// TIA Portal project "Tanque_PID" (V16)

(* hardware
DEVICE "S71500/ET200MP station_1"  S7-1500 station
   slot 0: "Perfil soporte_0"  Rack  6ES7 590-1***0-0AA0
   slot 1: "PLC_1"  CPU 1511-1 PN  6ES7 511-1AK02-0AB0  V2.5
      slot 3: "Display de la CPU_1"  6ES7591-1AA00-0AA0
      slot 32768: "Interfaz PROFINET_1"  X1
         slot 32769: "Puerto_1"  X1 P1
         slot 32770: "Puerto_2"  X1 P2
DEVICE "PC-System_1"  SIMATIC PC station
   slot 0: "Estación PC SIMATIC"  Rail  SIMATIC PC-Station  V1.0
      slot 125: "Stationmanager"  Station_Manager  V6.0.4
   slot 1: "HMI_RT_1"  WinCC RT Advanced  6AV2 104-0xxxx-xxxx  16.0.0.0
      slot 33792: "Interfaz del equipo"  Host interface
   slot 2: "IE general_1"  IE General  IE_CP  V8.2.0
*)

// ===== PLC "PLC_1"  CPU 1511-1 PN =====

VAR_GLOBAL   // PLC tag table "Tabla de variables estándar"
   "START_SISTEMA" AT %I0.0 : Bool;
   "STOP_SISTEMA" AT %I0.1 : Bool;
   "ENCENDIDO_SISTEMA" AT %M1.0 : Bool;
   "START_LIGHT" AT %Q0.0 : Bool;
   "STOP_LIGTH" AT %Q0.1 : Bool;
   "FILL_VALVE" AT %QW100 : Word;
   "DISCHARGE_VALVE" AT %QW102 : Word;
   "INPUT_FILL_VALVE" AT %MW10 : Word;
   "INPUT_DISCHARGE_VALVE" AT %MW12 : Word;
   "INPUT_FILL_VALVE_NORMAL" AT %MD14 : Real;
   "INPUT_DICHARGE_VALVE_NORMAL" AT %MD18 : Real;
   "DATA_INPUT_FILL_VALVE" AT %MW22 : Word;
   "DATA_INPUT_DISCHARGE_VALVE" AT %MW24 : Word;
   "CONTROL_MANUAL" AT %M1.1 : Bool;
   "CONTROL_AUTOMATICO_PID" AT %M1.2 : Bool;
   "LEVEL_METER" AT %IW100 : Word;
   "LEVEL_METER_NORMAL" AT %MD28 : Real;
   "LEVEL_METER_PANTALLA" AT %QW106 : Word;
   "INPUT_SP" AT %MW32 : Word;
   "SP_PANTALLA" AT %QW104 : Word;
   "SENSOR_NIVEL_INFERIOR" AT %I0.2 : Bool;
   "SENSOR_NIVEL_SUPERIOR" AT %I0.3 : Bool;
   "TANQUE_VACIO" AT %Q0.2 : Bool;
   "TANQUE_LLENO" AT %Q0.3 : Bool;
   "ON_PID_NIVEL" AT %M1.3 : Bool;
   "OFF_PID_NIVEL" AT %M1.4 : Bool;
   "PID_NIVEL" AT %M1.5 : Bool;
   "ON_PID_MANUAL" AT %M1.6 : Bool;
   "OFF_PID_MANUAL" AT %M1.7 : Bool;
   "PID_SET_MANUAL" AT %M2.0 : Bool;
   "DATA_PID_GAIN" AT %MD34 : Real;
   "DATA_PID_TI" AT %MD38 : Real;
   "DATA_PID_TD" AT %MD42 : Real;
   "OUT_PID_FILL_VALVE" AT %MW46 : Word;
   "INPUT_SP_PID" AT %MD48 : Real;
   "LEVEL_METER_PID" AT %MD54 : Real;
   "OUT_PID_FILL_VALVE_PID" AT %MD60 : Real;
   "START_SISTEMA_HMI" AT %M2.2 : Bool;
   "STOP_SISTEMA_HMI" AT %M2.3 : Bool;
   "CONTROL_MANUAL_CAUDAL" AT %M2.4 : Bool;
   "CONTROL_AUTOMATICO_PID_CAUDAL" AT %M2.5 : Bool;
   "CAUDAL_METER" AT %IW104 : Word;
   "CAUDAL_METER_NORMAL" AT %MD64 : Real;
   "CAUDAL_METER_PANTALLA" AT %QW110 : Word;
   "INPUT_SP_CAUDAL" AT %MW68 : Word;
   "SP_PANTALLA_CAUDAL" AT %QW112 : Word;
   "ON_PID_CAUDAL" AT %M2.6 : Bool;
   "OFF_PID_CAUDAL" AT %M2.7 : Bool;
   "PID_SET_MANUAL_CAUDAL" AT %M3.0 : Bool;
   "DATA_PID_GAIN_CAUDAL" AT %MD70 : Real;
   "DATA_PID_TI_CAUDAL" AT %MD74 : Real;
   "DATA_PID_TD_CAUDAL" AT %MD76 : Real;
   "INPUT_SP_PID_CAUDAL" AT %MD80 : Real;
   "CAUDAL_METER_PID" AT %MD84 : Real;
   "SENSOR_CAUDAL" AT %ID88 : Real;
   "OUT_PID_DISCHARGE_VALVE" AT %MW114 : Word;
   "OUT_PID_DISCHARGE_VALVE_PID" AT %MD92 : Real;
   "PID_CAUDAL" AT %M3.1 : Bool;
   "ON_PID_MANUAL_CAUDAL" AT %M3.2 : Bool;
   "OFF_PID_MANUAL_CAUDAL" AT %M3.3 : Bool;
   "PID_OUTPUT" AT %MD96 : Real;
   "ABS_PID_OUTPUT" AT %MD100 : Real;
   "SP_PANTALLA_MAS" AT %QW116 : Word;
   "SP_PANTALLA_MENOs" AT %QW118 : Word;
   "MITAD_VALVULA" AT %MD104 : Real;
   "50_VALVULA" AT %MW118 : Word;
   "PORCENT_CONEXION" AT %MD108 : Real;
   "PORCENT_NIVEL" AT %MD120 : Real;
   "PORCENT_NIVEL_INT" AT %MW122 : Word;
END_VAR

ORGANIZATION_BLOCK "1_Main"   // OB1, LAD, ProgramCycle
TITLE = "Main Program Sweep (Cycle)"
{ S7_Optimized_Access := 'TRUE' }
VERSION : 0.1
   VAR_INPUT
      Initial_Call : Bool;   // Initial call of this OB
      Remanence : Bool;   // =True, if remanent data are available
   END_VAR
   VAR_TEMP   // added for the SCL form of the ladder/FBD networks
      _w1 : Bool;
      _w2 : Bool;
      _w3 : Bool;
   END_VAR
BEGIN

REGION Network 1: ENCENDIDO Y APAGADO DEL SISTEMA
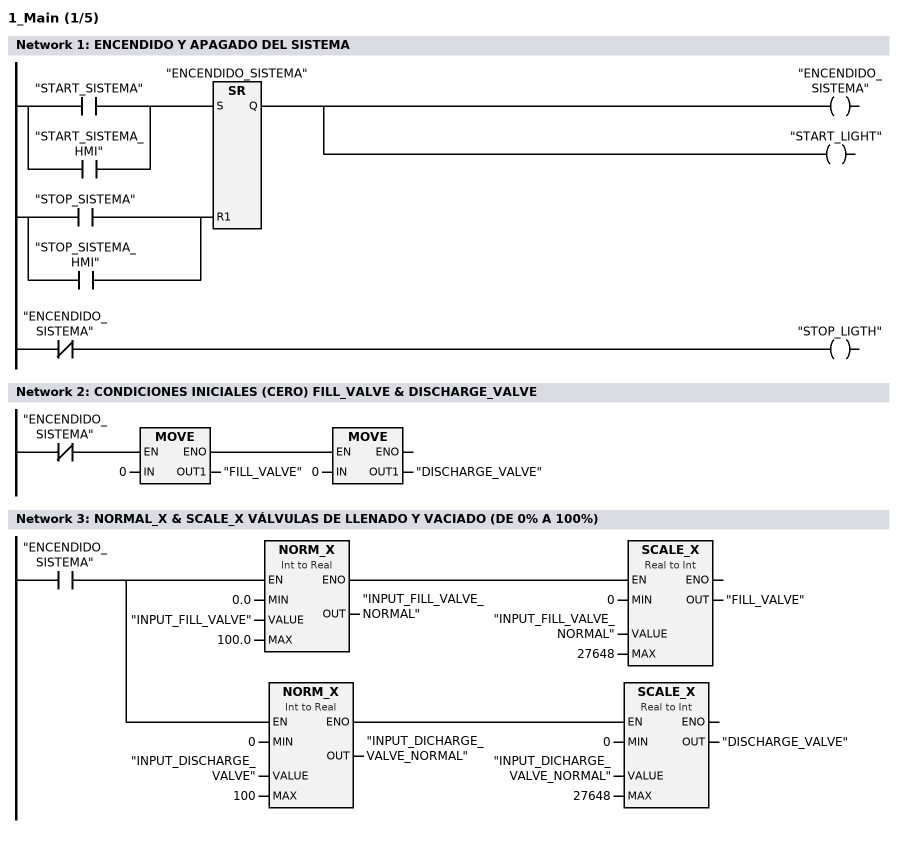
   RUNG wire#powerrail
      Contact( "START_SISTEMA" )
      wire#w1
      S_SR(operand := "ENCENDIDO_SISTEMA", r1 := wire#w2)
      wire#w3
      Coil( "ENCENDIDO_SISTEMA" )
   END_RUNG
   RUNG wire#powerrail
      Contact( "START_SISTEMA_HMI" )
   END_RUNG wire#w1
   RUNG wire#powerrail
      Contact( "STOP_SISTEMA" )
   END_RUNG wire#w2
   RUNG wire#powerrail
      Contact( "STOP_SISTEMA_HMI" )
   END_RUNG wire#w2
   RUNG wire#w3
      Coil( "START_LIGHT" )
   END_RUNG
   RUNG wire#powerrail
      I_Contact( "ENCENDIDO_SISTEMA" )
      Coil( "STOP_LIGTH" )
   END_RUNG
   // the same network as SCL:
   IF "START_SISTEMA" OR "START_SISTEMA_HMI" THEN
       "ENCENDIDO_SISTEMA" := TRUE;   // SR flip-flop
   END_IF;
   IF "STOP_SISTEMA" OR "STOP_SISTEMA_HMI" THEN "ENCENDIDO_SISTEMA" := FALSE; END_IF;
   #_w1 := "ENCENDIDO_SISTEMA";
   "ENCENDIDO_SISTEMA" := "ENCENDIDO_SISTEMA";
   "START_LIGHT" := #_w1;
   "STOP_LIGTH" := NOT "ENCENDIDO_SISTEMA";
END_REGION

REGION Network 2: CONDICIONES INICIALES (CERO) FILL_VALVE & DISCHARGE_VALVE
   RUNG wire#powerrail
      I_Contact( "ENCENDIDO_SISTEMA" )
      Move(in := 0, out1 => "FILL_VALVE")
      Move(in := 0, out1 => "DISCHARGE_VALVE")
   END_RUNG
   // the same network as SCL:
   IF NOT "ENCENDIDO_SISTEMA" THEN
       "FILL_VALVE" := 0;
       "DISCHARGE_VALVE" := 0;
   END_IF;
END_REGION

REGION Network 3: NORMAL_X & SCALE_X VÁLVULAS DE LLENADO Y VACIADO (DE 0% A 100%)
   RUNG wire#powerrail
      Contact( "ENCENDIDO_SISTEMA" )
      wire#w1
      { S7_Templates := "[SrcType := Int, DestType := Real]" } Normalize(min := 0.0, value := "INPUT_FILL_VALVE", max := 100.0, out => "INPUT_FILL_VALVE_NORMAL")
      { S7_Templates := "[SrcType := Real, DestType := Int]" } Scale(min := 0, value := "INPUT_FILL_VALVE_NORMAL", max := 27648, out => "FILL_VALVE")
   END_RUNG
   RUNG wire#w1
      { S7_Templates := "[SrcType := Int, DestType := Real]" } Normalize(min := 0, value := "INPUT_DISCHARGE_VALVE", max := 100, out => "INPUT_DICHARGE_VALVE_NORMAL")
      { S7_Templates := "[SrcType := Real, DestType := Int]" } Scale(min := 0, value := "INPUT_DICHARGE_VALVE_NORMAL", max := 27648, out => "DISCHARGE_VALVE")
   END_RUNG
   // the same network as SCL:
   IF "ENCENDIDO_SISTEMA" THEN
       "INPUT_FILL_VALVE_NORMAL" := NORM_X(MIN := 0.0, VALUE := "INPUT_FILL_VALVE", MAX := 100.0);
       "FILL_VALVE" := SCALE_X(MIN := 0, VALUE := "INPUT_FILL_VALVE_NORMAL", MAX := 27648);
       "INPUT_DICHARGE_VALVE_NORMAL" := NORM_X(MIN := 0, VALUE := "INPUT_DISCHARGE_VALVE", MAX := 100);
       "DISCHARGE_VALVE" := SCALE_X(MIN := 0, VALUE := "INPUT_DICHARGE_VALVE_NORMAL", MAX := 27648);
   END_IF;
END_REGION

REGION Network 4: CONTROL MANUAL & AUTOMÁTICO (PID_NIVEL)
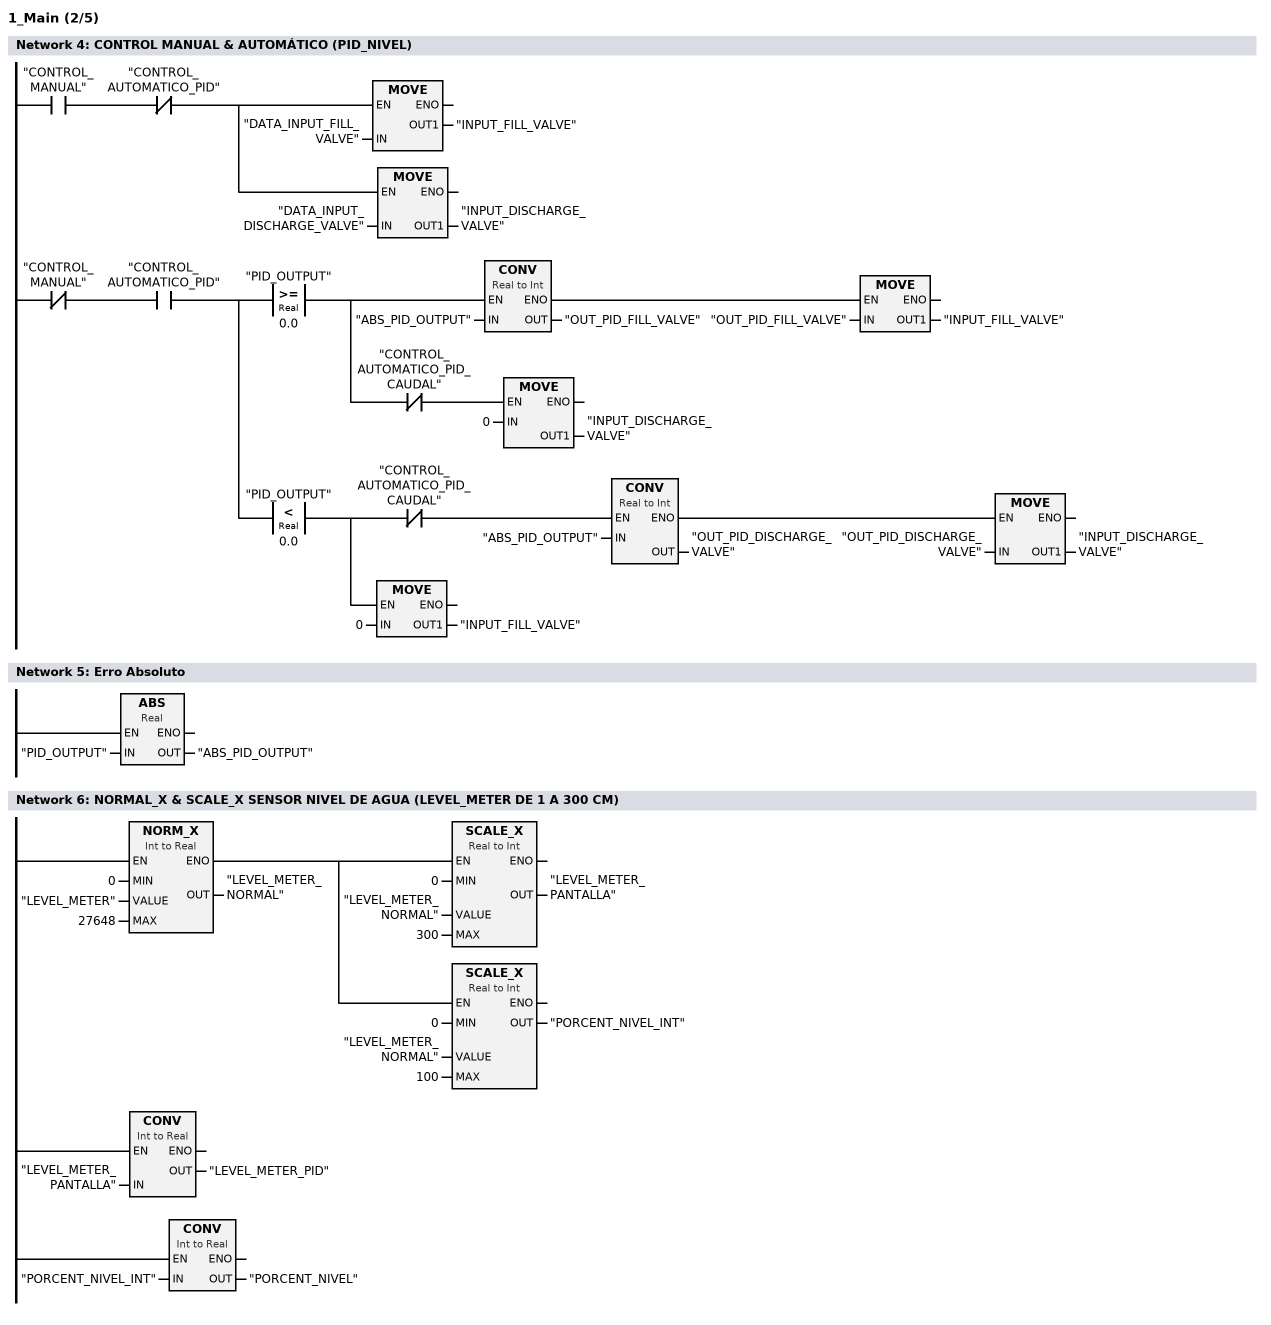
   RUNG wire#powerrail
      Contact( "CONTROL_MANUAL" )
      I_Contact( "CONTROL_AUTOMATICO_PID" )
      wire#w1
      Move(in := "DATA_INPUT_FILL_VALVE", out1 => "INPUT_FILL_VALVE")
   END_RUNG
   RUNG wire#w1
      Move(in := "DATA_INPUT_DISCHARGE_VALVE", out1 => "INPUT_DISCHARGE_VALVE")
   END_RUNG
   RUNG wire#powerrail
      I_Contact( "CONTROL_MANUAL" )
      Contact( "CONTROL_AUTOMATICO_PID" )
      wire#w2
      { S7_Templates := "SrcType := Real" } GE_Contact(in1 := "PID_OUTPUT", in2 := 0.0)
      wire#w3
      { S7_Templates := "[SrcType := Real, DestType := Int]" } Convert(in := "ABS_PID_OUTPUT", out => "OUT_PID_FILL_VALVE")
      Move(in := "OUT_PID_FILL_VALVE", out1 => "INPUT_FILL_VALVE")
   END_RUNG
   RUNG wire#w3
      I_Contact( "CONTROL_AUTOMATICO_PID_CAUDAL" )
      Move(in := 0, out1 => "INPUT_DISCHARGE_VALVE")
   END_RUNG
   RUNG wire#w2
      { S7_Templates := "SrcType := Real" } LT_Contact(in1 := "PID_OUTPUT", in2 := 0.0)
      wire#w4
      I_Contact( "CONTROL_AUTOMATICO_PID_CAUDAL" )
      { S7_Templates := "[SrcType := Real, DestType := Int]" } Convert(in := "ABS_PID_OUTPUT", out => "OUT_PID_DISCHARGE_VALVE")
      Move(in := "OUT_PID_DISCHARGE_VALVE", out1 => "INPUT_DISCHARGE_VALVE")
   END_RUNG
   RUNG wire#w4
      Move(in := 0, out1 => "INPUT_FILL_VALVE")
   END_RUNG
   // the same network as SCL:
   IF "CONTROL_MANUAL" AND NOT "CONTROL_AUTOMATICO_PID" THEN
       "INPUT_FILL_VALVE" := "DATA_INPUT_FILL_VALVE";
       "INPUT_DISCHARGE_VALVE" := "DATA_INPUT_DISCHARGE_VALVE";
   END_IF;
   #_w1 := NOT "CONTROL_MANUAL" AND "CONTROL_AUTOMATICO_PID";
   #_w2 := #_w1 AND ("PID_OUTPUT" >= 0.0);
   IF #_w2 THEN
       "OUT_PID_FILL_VALVE" := REAL_TO_INT("ABS_PID_OUTPUT");
       "INPUT_FILL_VALVE" := "OUT_PID_FILL_VALVE";
   END_IF;
   IF #_w2 AND NOT "CONTROL_AUTOMATICO_PID_CAUDAL" THEN "INPUT_DISCHARGE_VALVE" := 0; END_IF;
   #_w3 := #_w1 AND ("PID_OUTPUT" < 0.0);
   IF #_w3 AND NOT "CONTROL_AUTOMATICO_PID_CAUDAL" THEN
       "OUT_PID_DISCHARGE_VALVE" := REAL_TO_INT("ABS_PID_OUTPUT");
       "INPUT_DISCHARGE_VALVE" := "OUT_PID_DISCHARGE_VALVE";
   END_IF;
   IF #_w3 THEN "INPUT_FILL_VALVE" := 0; END_IF;
END_REGION

REGION Network 5: Erro Absoluto
   RUNG wire#powerrail
      { S7_Templates := "SrcType := Real" } Abs(in := "PID_OUTPUT", out => "ABS_PID_OUTPUT")
   END_RUNG
   // the same network as SCL:
   "ABS_PID_OUTPUT" := ABS("PID_OUTPUT");
END_REGION

REGION Network 6: NORMAL_X & SCALE_X SENSOR NIVEL DE AGUA (LEVEL_METER DE 1 A 300 CM)
   RUNG wire#powerrail
      { S7_Templates := "[SrcType := Int, DestType := Real]" } Normalize(min := 0, value := "LEVEL_METER", max := 27648, out => "LEVEL_METER_NORMAL")
      wire#w1
      { S7_Templates := "[SrcType := Real, DestType := Int]" } Scale(min := 0, value := "LEVEL_METER_NORMAL", max := 300, out => "LEVEL_METER_PANTALLA")
   END_RUNG
   RUNG wire#w1
      { S7_Templates := "[SrcType := Real, DestType := Int]" } Scale(min := 0, value := "LEVEL_METER_NORMAL", max := 100, out => "PORCENT_NIVEL_INT")
   END_RUNG
   RUNG wire#powerrail
      { S7_Templates := "[SrcType := Int, DestType := Real]" } Convert(in := "LEVEL_METER_PANTALLA", out => "LEVEL_METER_PID")
   END_RUNG
   RUNG wire#powerrail
      { S7_Templates := "[SrcType := Int, DestType := Real]" } Convert(in := "PORCENT_NIVEL_INT", out => "PORCENT_NIVEL")
   END_RUNG
   // the same network as SCL:
   "LEVEL_METER_NORMAL" := NORM_X(MIN := 0, VALUE := "LEVEL_METER", MAX := 27648);
   "LEVEL_METER_PANTALLA" := SCALE_X(MIN := 0, VALUE := "LEVEL_METER_NORMAL", MAX := 300);
   "PORCENT_NIVEL_INT" := SCALE_X(MIN := 0, VALUE := "LEVEL_METER_NORMAL", MAX := 100);
   "LEVEL_METER_PID" := INT_TO_REAL("LEVEL_METER_PANTALLA");
   "PORCENT_NIVEL" := INT_TO_REAL("PORCENT_NIVEL_INT");
END_REGION

REGION Network 7: INPUT_SP SP_PANTALLA
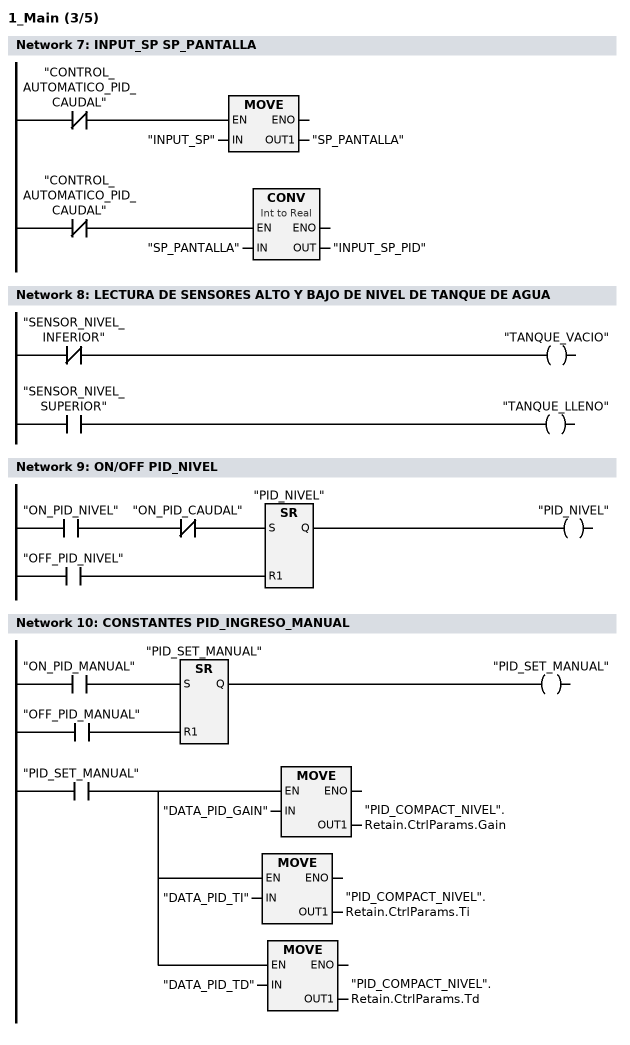
   RUNG wire#powerrail
      I_Contact( "CONTROL_AUTOMATICO_PID_CAUDAL" )
      Move(in := "INPUT_SP", out1 => "SP_PANTALLA")
   END_RUNG
   RUNG wire#powerrail
      I_Contact( "CONTROL_AUTOMATICO_PID_CAUDAL" )
      { S7_Templates := "[SrcType := Int, DestType := Real]" } Convert(in := "SP_PANTALLA", out => "INPUT_SP_PID")
   END_RUNG
   // the same network as SCL:
   IF NOT "CONTROL_AUTOMATICO_PID_CAUDAL" THEN
       "SP_PANTALLA" := "INPUT_SP";
       "INPUT_SP_PID" := INT_TO_REAL("SP_PANTALLA");
   END_IF;
END_REGION

REGION Network 8: LECTURA DE SENSORES ALTO Y BAJO DE NIVEL DE TANQUE DE AGUA
   RUNG wire#powerrail
      I_Contact( "SENSOR_NIVEL_INFERIOR" )
      Coil( "TANQUE_VACIO" )
   END_RUNG
   RUNG wire#powerrail
      Contact( "SENSOR_NIVEL_SUPERIOR" )
      Coil( "TANQUE_LLENO" )
   END_RUNG
   // the same network as SCL:
   "TANQUE_VACIO" := NOT "SENSOR_NIVEL_INFERIOR";
   "TANQUE_LLENO" := "SENSOR_NIVEL_SUPERIOR";
END_REGION

REGION Network 9: ON/OFF PID_NIVEL
   RUNG wire#powerrail
      Contact( "ON_PID_NIVEL" )
      I_Contact( "ON_PID_CAUDAL" )
      S_SR(operand := "PID_NIVEL", r1 := wire#w1)
      Coil( "PID_NIVEL" )
   END_RUNG
   RUNG wire#powerrail
      Contact( "OFF_PID_NIVEL" )
   END_RUNG wire#w1
   // the same network as SCL:
   IF "ON_PID_NIVEL" AND NOT "ON_PID_CAUDAL" THEN
       "PID_NIVEL" := TRUE;   // SR flip-flop
   END_IF;
   IF "OFF_PID_NIVEL" THEN "PID_NIVEL" := FALSE; END_IF;
   "PID_NIVEL" := "PID_NIVEL";
END_REGION

REGION Network 10: CONSTANTES PID_INGRESO_MANUAL
   RUNG wire#powerrail
      Contact( "ON_PID_MANUAL" )
      S_SR(operand := "PID_SET_MANUAL", r1 := wire#w1)
      Coil( "PID_SET_MANUAL" )
   END_RUNG
   RUNG wire#powerrail
      Contact( "OFF_PID_MANUAL" )
   END_RUNG wire#w1
   RUNG wire#powerrail
      Contact( "PID_SET_MANUAL" )
      wire#w2
      Move(in := "DATA_PID_GAIN", out1 => "PID_COMPACT_NIVEL".Retain.CtrlParams.Gain)
   END_RUNG
   RUNG wire#w2
      Move(in := "DATA_PID_TI", out1 => "PID_COMPACT_NIVEL".Retain.CtrlParams.Ti)
   END_RUNG
   RUNG wire#w2
      Move(in := "DATA_PID_TD", out1 => "PID_COMPACT_NIVEL".Retain.CtrlParams.Td)
   END_RUNG
   // the same network as SCL:
   IF "ON_PID_MANUAL" THEN
       "PID_SET_MANUAL" := TRUE;   // SR flip-flop
   END_IF;
   IF "OFF_PID_MANUAL" THEN "PID_SET_MANUAL" := FALSE; END_IF;
   "PID_SET_MANUAL" := "PID_SET_MANUAL";
   IF "PID_SET_MANUAL" THEN
       "PID_COMPACT_NIVEL".Retain.CtrlParams.Gain := "DATA_PID_GAIN";
       "PID_COMPACT_NIVEL".Retain.CtrlParams.Ti := "DATA_PID_TI";
       "PID_COMPACT_NIVEL".Retain.CtrlParams.Td := "DATA_PID_TD";
   END_IF;
END_REGION

REGION Network 11: CONTROL MANUAL & AUTOMÁTICO (PID_CAUDAL)
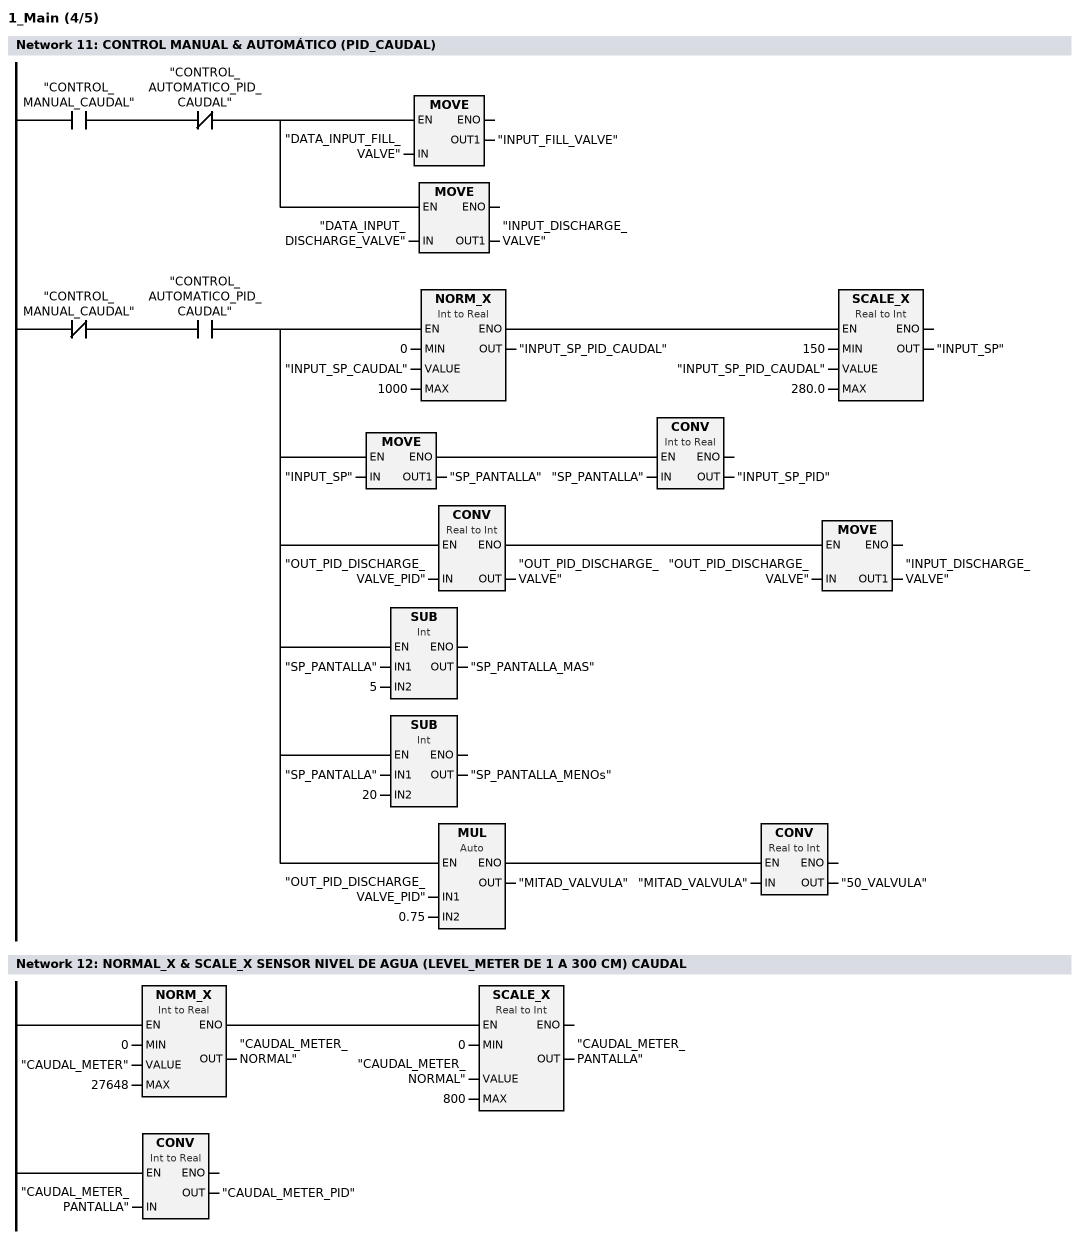
   RUNG wire#powerrail
      Contact( "CONTROL_MANUAL_CAUDAL" )
      I_Contact( "CONTROL_AUTOMATICO_PID_CAUDAL" )
      wire#w1
      Move(in := "DATA_INPUT_FILL_VALVE", out1 => "INPUT_FILL_VALVE")
   END_RUNG
   RUNG wire#w1
      Move(in := "DATA_INPUT_DISCHARGE_VALVE", out1 => "INPUT_DISCHARGE_VALVE")
   END_RUNG
   RUNG wire#powerrail
      I_Contact( "CONTROL_MANUAL_CAUDAL" )
      Contact( "CONTROL_AUTOMATICO_PID_CAUDAL" )
      wire#w2
      { S7_Templates := "[SrcType := Int, DestType := Real]" } Normalize(min := 0, value := "INPUT_SP_CAUDAL", max := 1000, out => "INPUT_SP_PID_CAUDAL")
      { S7_Templates := "[SrcType := Real, DestType := Int]" } Scale(min := 150, value := "INPUT_SP_PID_CAUDAL", max := 280.0, out => "INPUT_SP")
   END_RUNG
   RUNG wire#w2
      Move(in := "INPUT_SP", out1 => "SP_PANTALLA")
      { S7_Templates := "[SrcType := Int, DestType := Real]" } Convert(in := "SP_PANTALLA", out => "INPUT_SP_PID")
   END_RUNG
   RUNG wire#w2
      { S7_Templates := "[SrcType := Real, DestType := Int]" } Convert(in := "OUT_PID_DISCHARGE_VALVE_PID", out => "OUT_PID_DISCHARGE_VALVE")
      Move(in := "OUT_PID_DISCHARGE_VALVE", out1 => "INPUT_DISCHARGE_VALVE")
   END_RUNG
   RUNG wire#w2
      { S7_Templates := "SrcType := Int" } Sub(in1 := "SP_PANTALLA", in2 := 5, out => "SP_PANTALLA_MAS")
   END_RUNG
   RUNG wire#w2
      { S7_Templates := "SrcType := Int" } Sub(in1 := "SP_PANTALLA", in2 := 20, out => "SP_PANTALLA_MENOs")
   END_RUNG
   RUNG wire#w2
      Mul(in1 := "OUT_PID_DISCHARGE_VALVE_PID", in2 := 0.75, out => "MITAD_VALVULA")
      { S7_Templates := "[SrcType := Real, DestType := Int]" } Convert(in := "MITAD_VALVULA", out => "50_VALVULA")
   END_RUNG
   // the same network as SCL:
   IF "CONTROL_MANUAL_CAUDAL" AND NOT "CONTROL_AUTOMATICO_PID_CAUDAL" THEN
       "INPUT_FILL_VALVE" := "DATA_INPUT_FILL_VALVE";
       "INPUT_DISCHARGE_VALVE" := "DATA_INPUT_DISCHARGE_VALVE";
   END_IF;
   IF NOT "CONTROL_MANUAL_CAUDAL" AND "CONTROL_AUTOMATICO_PID_CAUDAL" THEN
       "INPUT_SP_PID_CAUDAL" := NORM_X(MIN := 0, VALUE := "INPUT_SP_CAUDAL", MAX := 1000);
       "INPUT_SP" := SCALE_X(MIN := 150, VALUE := "INPUT_SP_PID_CAUDAL", MAX := 280.0);
       "SP_PANTALLA" := "INPUT_SP";
       "INPUT_SP_PID" := INT_TO_REAL("SP_PANTALLA");
       "OUT_PID_DISCHARGE_VALVE" := REAL_TO_INT("OUT_PID_DISCHARGE_VALVE_PID");
       "INPUT_DISCHARGE_VALVE" := "OUT_PID_DISCHARGE_VALVE";
       "SP_PANTALLA_MAS" := "SP_PANTALLA" - 5;
       "SP_PANTALLA_MENOs" := "SP_PANTALLA" - 20;
       "MITAD_VALVULA" := "OUT_PID_DISCHARGE_VALVE_PID" * 0.75;
       "50_VALVULA" := REAL_TO_INT("MITAD_VALVULA");
   END_IF;
END_REGION

REGION Network 12: NORMAL_X & SCALE_X SENSOR NIVEL DE AGUA (LEVEL_METER DE 1 A 300 CM) CAUDAL
   RUNG wire#powerrail
      { S7_Templates := "[SrcType := Int, DestType := Real]" } Normalize(min := 0, value := "CAUDAL_METER", max := 27648, out => "CAUDAL_METER_NORMAL")
      { S7_Templates := "[SrcType := Real, DestType := Int]" } Scale(min := 0, value := "CAUDAL_METER_NORMAL", max := 800, out => "CAUDAL_METER_PANTALLA")
   END_RUNG
   RUNG wire#powerrail
      { S7_Templates := "[SrcType := Int, DestType := Real]" } Convert(in := "CAUDAL_METER_PANTALLA", out => "CAUDAL_METER_PID")
   END_RUNG
   // the same network as SCL:
   "CAUDAL_METER_NORMAL" := NORM_X(MIN := 0, VALUE := "CAUDAL_METER", MAX := 27648);
   "CAUDAL_METER_PANTALLA" := SCALE_X(MIN := 0, VALUE := "CAUDAL_METER_NORMAL", MAX := 800);
   "CAUDAL_METER_PID" := INT_TO_REAL("CAUDAL_METER_PANTALLA");
END_REGION

REGION Network 13: INPUT_SP CAUDAL SP_PANTALLA
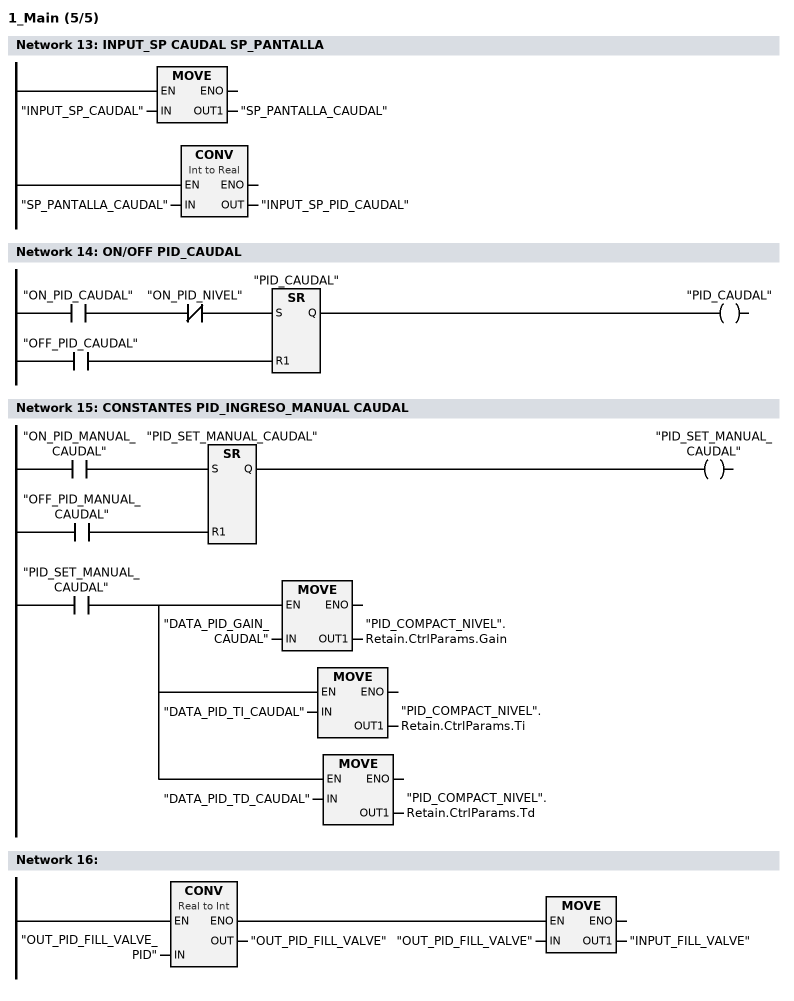
   RUNG wire#powerrail
      Move(in := "INPUT_SP_CAUDAL", out1 => "SP_PANTALLA_CAUDAL")
   END_RUNG
   RUNG wire#powerrail
      { S7_Templates := "[SrcType := Int, DestType := Real]" } Convert(in := "SP_PANTALLA_CAUDAL", out => "INPUT_SP_PID_CAUDAL")
   END_RUNG
   // the same network as SCL:
   "SP_PANTALLA_CAUDAL" := "INPUT_SP_CAUDAL";
   "INPUT_SP_PID_CAUDAL" := INT_TO_REAL("SP_PANTALLA_CAUDAL");
END_REGION

REGION Network 14: ON/OFF PID_CAUDAL
   RUNG wire#powerrail
      Contact( "ON_PID_CAUDAL" )
      I_Contact( "ON_PID_NIVEL" )
      S_SR(operand := "PID_CAUDAL", r1 := wire#w1)
      Coil( "PID_CAUDAL" )
   END_RUNG
   RUNG wire#powerrail
      Contact( "OFF_PID_CAUDAL" )
   END_RUNG wire#w1
   // the same network as SCL:
   IF "ON_PID_CAUDAL" AND NOT "ON_PID_NIVEL" THEN
       "PID_CAUDAL" := TRUE;   // SR flip-flop
   END_IF;
   IF "OFF_PID_CAUDAL" THEN "PID_CAUDAL" := FALSE; END_IF;
   "PID_CAUDAL" := "PID_CAUDAL";
END_REGION

REGION Network 15: CONSTANTES PID_INGRESO_MANUAL CAUDAL
   RUNG wire#powerrail
      Contact( "ON_PID_MANUAL_CAUDAL" )
      S_SR(operand := "PID_SET_MANUAL_CAUDAL", r1 := wire#w1)
      Coil( "PID_SET_MANUAL_CAUDAL" )
   END_RUNG
   RUNG wire#powerrail
      Contact( "OFF_PID_MANUAL_CAUDAL" )
   END_RUNG wire#w1
   RUNG wire#powerrail
      Contact( "PID_SET_MANUAL_CAUDAL" )
      wire#w2
      Move(in := "DATA_PID_GAIN_CAUDAL", out1 => "PID_COMPACT_NIVEL".Retain.CtrlParams.Gain)
   END_RUNG
   RUNG wire#w2
      Move(in := "DATA_PID_TI_CAUDAL", out1 => "PID_COMPACT_NIVEL".Retain.CtrlParams.Ti)
   END_RUNG
   RUNG wire#w2
      Move(in := "DATA_PID_TD_CAUDAL", out1 => "PID_COMPACT_NIVEL".Retain.CtrlParams.Td)
   END_RUNG
   // the same network as SCL:
   IF "ON_PID_MANUAL_CAUDAL" THEN
       "PID_SET_MANUAL_CAUDAL" := TRUE;   // SR flip-flop
   END_IF;
   IF "OFF_PID_MANUAL_CAUDAL" THEN "PID_SET_MANUAL_CAUDAL" := FALSE; END_IF;
   "PID_SET_MANUAL_CAUDAL" := "PID_SET_MANUAL_CAUDAL";
   IF "PID_SET_MANUAL_CAUDAL" THEN
       "PID_COMPACT_NIVEL".Retain.CtrlParams.Gain := "DATA_PID_GAIN_CAUDAL";
       "PID_COMPACT_NIVEL".Retain.CtrlParams.Ti := "DATA_PID_TI_CAUDAL";
       "PID_COMPACT_NIVEL".Retain.CtrlParams.Td := "DATA_PID_TD_CAUDAL";
   END_IF;
END_REGION

REGION Network 16
   RUNG wire#powerrail
      { S7_Templates := "[SrcType := Real, DestType := Int]" } Convert(in := "OUT_PID_FILL_VALVE_PID", out => "OUT_PID_FILL_VALVE")
      Move(in := "OUT_PID_FILL_VALVE", out1 => "INPUT_FILL_VALVE")
   END_RUNG
   // the same network as SCL:
   "OUT_PID_FILL_VALVE" := REAL_TO_INT("OUT_PID_FILL_VALVE_PID");
   "INPUT_FILL_VALVE" := "OUT_PID_FILL_VALVE";
END_REGION
END_ORGANIZATION_BLOCK

ORGANIZATION_BLOCK "2_Nivel_PID"   // OB30, LAD, CyclicInterrupt
{ S7_Optimized_Access := 'TRUE' }
VERSION : 0.1
   VAR_INPUT
      Initial_Call : Bool;   // Initial call of this OB
      Event_Count : Int;   // Events discarded
   END_VAR
   VAR_TEMP   // added for the SCL form of the ladder/FBD networks
      _w1 : Bool;
   END_VAR
BEGIN

REGION Network 1
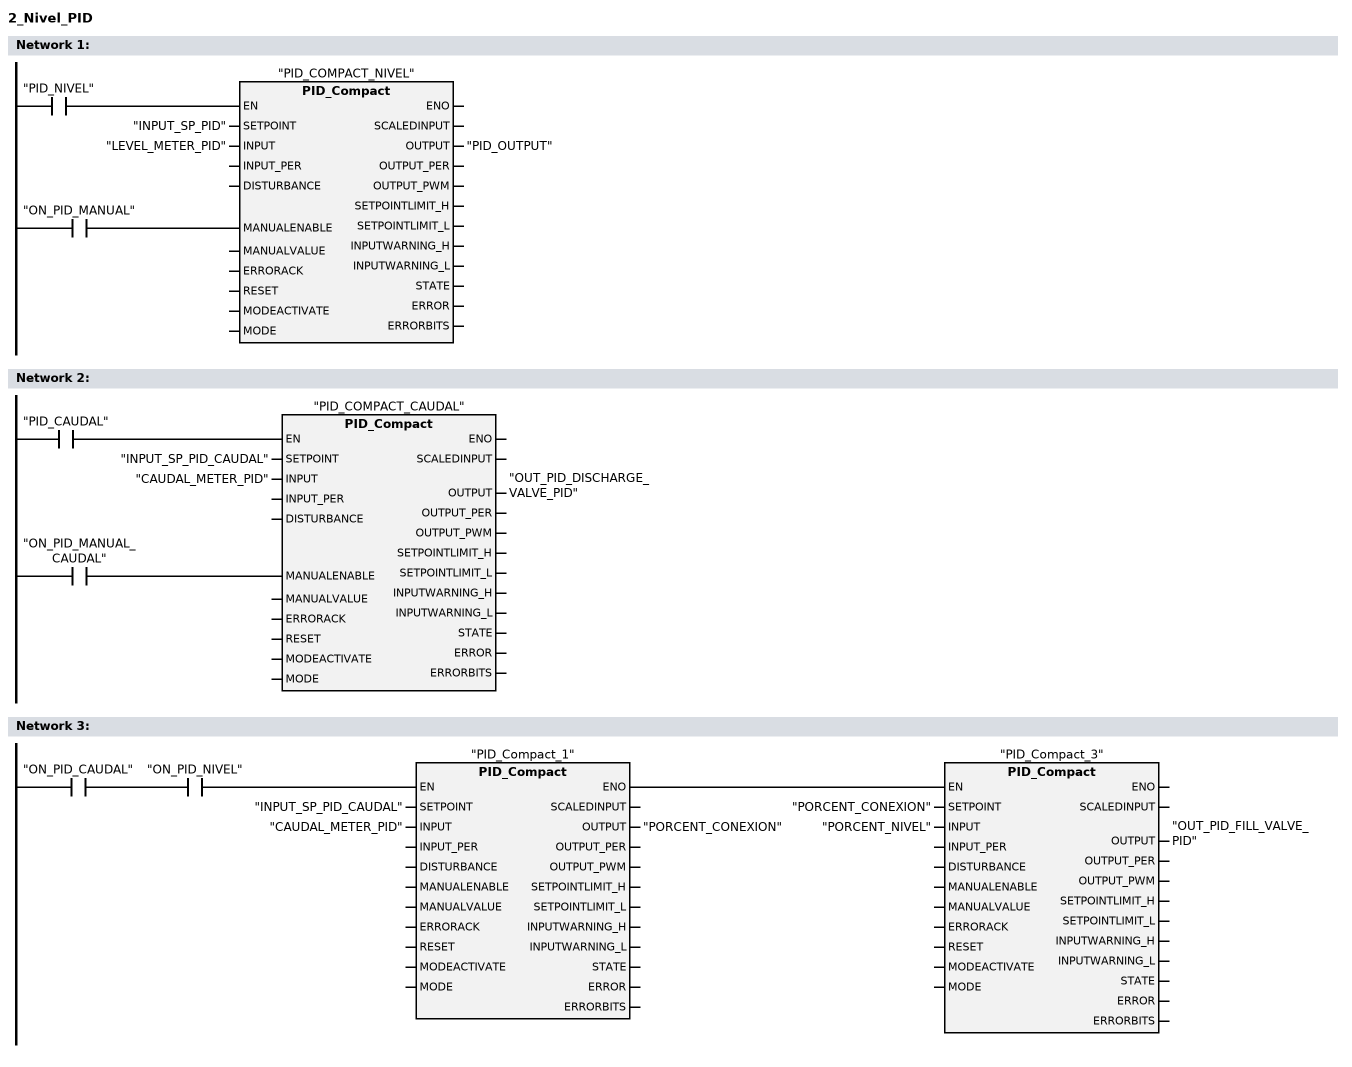
   IF "PID_NIVEL" THEN
       "PID_COMPACT_NIVEL"(Setpoint := "INPUT_SP_PID",   // PID_Compact
                           Input := "LEVEL_METER_PID",
                           ManualEnable := "ON_PID_MANUAL",
                           Output => "PID_OUTPUT");
   END_IF;
END_REGION

REGION Network 2
   IF "PID_CAUDAL" THEN
       "PID_COMPACT_CAUDAL"(Setpoint := "INPUT_SP_PID_CAUDAL",   // PID_Compact
                            Input := "CAUDAL_METER_PID",
                            ManualEnable := "ON_PID_MANUAL_CAUDAL",
                            Output => "OUT_PID_DISCHARGE_VALVE_PID");
   END_IF;
END_REGION

REGION Network 3
   // ENO of a box is taken as its EN; it also drops when the box reports an error
   #_w1 := "ON_PID_CAUDAL" AND "ON_PID_NIVEL";
   IF #_w1 THEN
       "PID_Compact_1"(Setpoint := "INPUT_SP_PID_CAUDAL", Input := "CAUDAL_METER_PID", Output => "PORCENT_CONEXION");   // PID_Compact
       "PID_Compact_3"(Setpoint := "PORCENT_CONEXION", Input := "PORCENT_NIVEL", Output => "OUT_PID_FILL_VALVE_PID");   // PID_Compact
   END_IF;
END_REGION
END_ORGANIZATION_BLOCK

(* ===== HMI "HMI_RT_1" =====
system functions are stored by id; their names below are inferred from use
connection "HMI_Conexión_1": ETHERNET, S7_1500_OMS

HMI tags "Tabla de variables estándar"
   "DATA_INPUT_FILL_VALVE" : Word = PLC DATA_INPUT_FILL_VALVE AT %MW22, 1 s
   "DATA_INPUT_DISCHARGE_VALVE" : Word = PLC DATA_INPUT_DISCHARGE_VALVE AT %MW24, 1 s
   "START_SISTEMA" : Bool = PLC START_SISTEMA AT %I0.0, 1 s
   "STOP_SISTEMA" : Bool = PLC STOP_SISTEMA AT %I0.1, 1 s
   "ENCENDIDO_SISTEMA" : Bool = PLC ENCENDIDO_SISTEMA AT %M1.0, 1 s
   "STOP_LIGTH" : Bool = PLC STOP_LIGTH AT %Q0.1, 1 s
   "START_LIGHT" : Bool = PLC START_LIGHT AT %Q0.0, 1 s
   "LEVEL_METER" : Word = PLC LEVEL_METER AT %IW100, 1 s
   "LEVEL_METER_PANTALLA" : Word = PLC LEVEL_METER_PANTALLA AT %QW106, 1 s
   "START_SISTEMA_HMI" : Bool = PLC START_SISTEMA_HMI AT %M2.2, 1 s
   "STOP_SISTEMA_HMI" : Bool = PLC STOP_SISTEMA_HMI AT %M2.3, 1 s
   "CONTROL_MANUAL" : Bool = PLC CONTROL_MANUAL AT %M1.1, 1 s
   "CONTROL_AUTOMATICO_PID" : Bool = PLC CONTROL_AUTOMATICO_PID AT %M1.2, 1 s
   "INPUT_SP" : Word = PLC INPUT_SP AT %MW32, 1 s
   "ON_PID_NIVEL" : Bool = PLC ON_PID_NIVEL AT %M1.3, 1 s
   "OFF_PID_NIVEL" : Bool = PLC OFF_PID_NIVEL AT %M1.4, 1 s
   "OUT_PID_FILL_VALVE_PID" : Real = PLC OUT_PID_FILL_VALVE_PID AT %MD60, 1 s
   "DATA_PID_GAIN" : Real = PLC DATA_PID_GAIN AT %MD34, 1 s
   "DATA_PID_TI" : Real = PLC DATA_PID_TI AT %MD38, 1 s
   "DATA_PID_TD" : Real = PLC DATA_PID_TD AT %MD42, 1 s
   "INPUT_SP_PID" : Real = PLC INPUT_SP_PID AT %MD48, 1 s
   "CONTROL_MANUAL_CAUDAL" : Bool = PLC CONTROL_MANUAL_CAUDAL AT %M2.4, 1 s
   "CONTROL_AUTOMATICO_PID_CAUDAL" : Bool = PLC CONTROL_AUTOMATICO_PID_CAUDAL AT %M2.5, 1 s
   "INPUT_SP_CAUDAL" : Word = PLC INPUT_SP_CAUDAL AT %MW68, 1 s
   "ON_PID_CAUDAL" : Bool = PLC ON_PID_CAUDAL AT %M2.6, 1 s
   "OFF_PID_CAUDAL" : Bool = PLC OFF_PID_CAUDAL AT %M2.7, 1 s
   "DATA_PID_GAIN_CAUDAL" : Real = PLC DATA_PID_GAIN_CAUDAL AT %MD70, 1 s
   "DATA_PID_TI_CAUDAL" : Real = PLC DATA_PID_TI_CAUDAL AT %MD74, 1 s
   "DATA_PID_TD_CAUDAL" : Real = PLC DATA_PID_TD_CAUDAL AT %MD76, 1 s
   "INPUT_SP_PID_CAUDAL" : Real = PLC INPUT_SP_PID_CAUDAL AT %MD80, 1 s
   "CAUDAL_METER_PID" : Real = PLC CAUDAL_METER_PID AT %MD84, 1 s
   "OUT_PID_DISCHARGE_VALVE_PID" : Real = PLC OUT_PID_DISCHARGE_VALVE_PID AT %MD92, 1 s
   "CAUDAL_METER_PANTALLA" : Word = PLC CAUDAL_METER_PANTALLA AT %QW110, 1 s
   "ON_PID_MANUAL_CAUDAL" : Bool = PLC ON_PID_MANUAL_CAUDAL AT %M3.2, 1 s
   "ON_PID_MANUAL" : Bool = PLC ON_PID_MANUAL AT %M1.6, 1 s
   "SP_PANTALLA" : Word = PLC SP_PANTALLA AT %QW104, 1 s
   "SP_PANTALLA_CAUDAL" : Word = PLC SP_PANTALLA_CAUDAL AT %QW112, 1 s
   "INPUT_FILL_VALVE" : Word = PLC INPUT_FILL_VALVE AT %MW10, 1 s
   "ABS_PID_OUTPUT" : Real = PLC ABS_PID_OUTPUT AT %MD100, 1 s
   "PORCENT_NIVEL" : Real = PLC PORCENT_NIVEL AT %MD120, 1 s
   "PORCENT_CONEXION" : Real = PLC PORCENT_CONEXION AT %MD108, 1 s

screen "1_Carátula" 1024x768
   Button "Botón_1" at 569,711 size 121x46; TextOff 'Control Nivel'
      on Click: ActivateScreen("3_Control_Nivel", 0)
   Button "Botón_5" at 869,712 size 126x46; TextOff 'Ir a Curvas'
      on Click: ActivateScreen("4_Curvas_Nivel", 0)
   Button "Botón_2" at 716,711 size 130x46; TextOff 'Control Caudal'
      on Click: ActivateScreen("2_Control_Caudal", 0)
   Button "Botón_3" at 362,712 size 187x46; TextOff 'Control General Caudal'
      on Click: ActivateScreen("6_Control_General", 0)

screen "2_Control_Caudal" 1024x768
   GraphicView "Visor de gráficos_2" at 1,0 size 1023x766; Picture "Gráfico_22"
   GraphicView "Visor de gráficos_1" at 0,0 size 574x768; Picture "steven_tanque_png"
   Bar "Barra_1" at 261,226 size 72x397; MinimumValue 0; MaximumValue 300
      ProcessValue <- "LEVEL_METER_PANTALLA"
   Button "Botón_1" at 603,24 size 125x34; TextOff 'Start_Sistema'
      on Press: SetBit("START_SISTEMA_HMI")
      on Release: ResetBit("START_SISTEMA_HMI")
   Button "Botón_2" at 811,26 size 123x32; TextOff 'Stop_Sistema'
      on Release: ResetBit("STOP_SISTEMA_HMI")
      on Press: SetBit("STOP_SISTEMA_HMI")
   IOField "Campo ES_2" at 752,158 size 59x39; FormatPattern 999
      ProcessValue <- "DATA_INPUT_DISCHARGE_VALVE"
   TextField "Campo de texto_2" at 703,127 size 175x25; Text '% Válvula de Salida'
   Circle "Círculo_1" at 651,64 size 46x46
      Appearance <- "START_LIGHT"
   Circle "Círculo_2" at 846,65 size 45x45
      Appearance <- "STOP_LIGTH"
   Switch "Interruptor_1" at 610,213 size 133x56; CaptionText 'Control Manual'; TextOff 'OFF'; TextOn 'ON'
      ProcessValue <- "CONTROL_MANUAL_CAUDAL"
   Switch "Interruptor_2" at 799,213 size 161x56; TextOn 'ON'; CaptionText 'Control Automático'; TextOff 'OFF'
      ProcessValue <- "CONTROL_AUTOMATICO_PID_CAUDAL"
   IOField "Campo ES_3" at 643,325 size 60x40; FormatPattern 999
      ProcessValue <- "INPUT_SP_CAUDAL"
   TextField "Campo de texto_3" at 610,295 size 127x25; Text 'Valor SetPoint'
   Button "Botón_3" at 799,301 size 137x33; TextOff 'ON_PID_Caudal'
      on Release: ResetBit("ON_PID_CAUDAL")
      on Press: SetBit("ON_PID_CAUDAL")
   Button "Botón_4" at 799,345 size 139x36; TextOff 'OFF_PID_Caudal'
      on Release: ResetBit("OFF_PID_NIVEL")
      on Press: SetBit("OFF_PID_CAUDAL")
   Button "Botón_5" at 762,697 size 116x50; TextOff 'Ir a Curvas'
      on Click: ActivateScreen("4_Curvas_Nivel", 0)
   Button "Botón_6" at 891,695 size 116x50; TextOff 'Ir a Inicio'
      on Click: ActivateScreen("1_Carátula", 0)
   IOField "Campo ES_5" at 607,561 size 60x40; FormatPattern 999
      ProcessValue <- "INPUT_SP_PID_CAUDAL"
   IOField "Campo ES_6" at 608,616 size 59x40; FormatPattern 999
      ProcessValue <- "CAUDAL_METER_PANTALLA"
   IOField "Campo ES_7" at 864,595 size 132x40
      ProcessValue <- "OUT_PID_DISCHARGE_VALVE_PID"
   GraphicView "Visor de gráficos_3" at 723,570 size 98x90; Picture "Gráfico_23"
   TextField "Campo de texto_5" at 611,655 size 53x25; Text 'Input'
   TextField "Campo de texto_6" at 903,564 size 65x25; Text 'Output'
   TextField "Campo de texto_7" at 601,536 size 78x25; Text 'Setpoint'
   IOField "Campo ES_4" at 814,457 size 129x34
      ProcessValue <- "DATA_PID_TI_CAUDAL"
   IOField "Campo ES_8" at 814,499 size 130x34
      ProcessValue <- "DATA_PID_TD_CAUDAL"
   IOField "Campo ES_9" at 814,413 size 130x35
      ProcessValue <- "DATA_PID_GAIN_CAUDAL"
   Switch "Interruptor_3" at 585,427 size 165x56; TextOn 'ON'; CaptionText 'Control Manual PID'; TextOff 'OFF'
      ProcessValue <- "ON_PID_MANUAL_CAUDAL"
   TextField "Campo de texto_4" at 776,417 size 28x25; Text 'Kp'
   TextField "Campo de texto_8" at 779,463 size 20x25; Text 'Ti'
   TextField "Campo de texto_9" at 779,503 size 26x25; Text 'Td'
   TextField "Campo de texto_10" at 174,33 size 241x43; Text 'Control Caudal'
   Button "Botón_7" at 629,697 size 121x48; TextOff 'Control Nivel'
      on Click: ActivateScreen("3_Control_Nivel", 0)

screen "4_Curvas_Nivel" 1024x768
   TrendView "Visor de curvas_1" at 11,4 size 998x388
   Button "Botón_1" at 893,714 size 116x50; TextOff 'Ir a Control'
      on Click: ActivateScreen("2_Control_Caudal", 0)
   Button "Botón_2" at 767,714 size 116x50; TextOff 'Ir a Inicio'
      on Click: ActivateScreen("1_Carátula", 0)
   TrendView "Visor de curvas_2" at 20,399 size 989x309

screen "3_Control_Nivel" 1024x768
   GraphicView "Visor de gráficos_2" at 1,0 size 1023x766; Picture "Gráfico_22"
   GraphicView "Visor de gráficos_1" at 0,0 size 574x768; Picture "steven_tanque_png"
   Bar "Barra_1" at 261,226 size 72x397; MinimumValue 0; MaximumValue 300
      ProcessValue <- "LEVEL_METER_PANTALLA"
   Button "Botón_1" at 603,27 size 125x31; TextOff 'Start_Sistema'
      on Release: ResetBit("START_SISTEMA_HMI")
      on Press: SetBit("START_SISTEMA_HMI")
   Button "Botón_2" at 811,26 size 123x32; TextOff 'Stop_Sistema'
      on Release: ResetBit("STOP_SISTEMA_HMI")
      on Press: SetBit("STOP_SISTEMA_HMI")
   IOField "Campo ES_1" at 643,161 size 60x39; FormatPattern 999
      ProcessValue <- "DATA_INPUT_FILL_VALVE"
   IOField "Campo ES_2" at 846,161 size 59x39; FormatPattern 999
      ProcessValue <- "DATA_INPUT_DISCHARGE_VALVE"
   TextField "Campo de texto_1" at 573,130 size 189x25; Text '% Válvula de Entrada'
   TextField "Campo de texto_2" at 781,126 size 175x25; Text '% Válvula de Salida'
   Circle "Círculo_1" at 651,64 size 46x46
      Appearance <- "START_LIGHT"
   Circle "Círculo_2" at 846,65 size 45x45
      Appearance <- "STOP_LIGTH"
   Switch "Interruptor_1" at 610,213 size 133x56; TextOn 'ON'; CaptionText 'Control Manual'; TextOff 'OFF'
      ProcessValue <- "CONTROL_MANUAL"
   Switch "Interruptor_2" at 799,213 size 161x56; TextOn 'ON'; CaptionText 'Control Automático'; TextOff 'OFF'
      ProcessValue <- "CONTROL_AUTOMATICO_PID"
   IOField "Campo ES_3" at 643,325 size 60x40; FormatPattern 999
      ProcessValue <- "INPUT_SP"
   TextField "Campo de texto_3" at 610,295 size 127x25; Text 'Valor SetPoint'
   Button "Botón_3" at 799,301 size 131x33; TextOff 'ON_PID_Nivel'
      on Release: ResetBit("ON_PID_NIVEL")
      on Press: SetBit("ON_PID_NIVEL")
   Button "Botón_4" at 799,345 size 131x33; TextOff 'OFF_PID_Nivel'
      on Release: ResetBit("OFF_PID_NIVEL")
      on Press: SetBit("OFF_PID_NIVEL")
   Button "Botón_5" at 762,697 size 116x49; TextOff 'Ir a Curvas'
      on Click: ActivateScreen("4_Curvas_Nivel", 0)
   Button "Botón_6" at 891,696 size 116x50; TextOff 'Ir a Inicio'
      on Click: ActivateScreen("1_Carátula", 0)
   IOField "Campo ES_5" at 607,561 size 60x40; FormatPattern 999
      ProcessValue <- "INPUT_SP_PID"
   IOField "Campo ES_6" at 608,616 size 59x40; FormatPattern 99999
      ProcessValue <- "LEVEL_METER_PANTALLA"
   IOField "Campo ES_7" at 864,595 size 132x40; FormatPattern s999.999
      ProcessValue <- "ABS_PID_OUTPUT"
   GraphicView "Visor de gráficos_3" at 723,570 size 98x90; Picture "Gráfico_23"
   TextField "Campo de texto_5" at 611,655 size 53x25; Text 'Input'
   TextField "Campo de texto_6" at 903,564 size 65x25; Text 'Output'
   TextField "Campo de texto_7" at 601,536 size 78x25; Text 'Setpoint'
   IOField "Campo ES_4" at 814,457 size 129x34; FormatPattern s999.999
      ProcessValue <- "DATA_PID_TI"
   IOField "Campo ES_8" at 814,499 size 130x34; FormatPattern s999.999
      ProcessValue <- "DATA_PID_TD"
   IOField "Campo ES_9" at 814,413 size 130x35; FormatPattern s999.999
      ProcessValue <- "DATA_PID_GAIN"
   Switch "Interruptor_3" at 607,427 size 133x56; TextOn 'ON'; CaptionText 'Control Manual'; TextOff 'OFF'
      ProcessValue <- "ON_PID_MANUAL"
   TextField "Campo de texto_4" at 776,417 size 28x25; Text 'Kp'
   TextField "Campo de texto_8" at 779,463 size 20x25; Text 'Ti'
   TextField "Campo de texto_9" at 779,503 size 26x25; Text 'Td'
   TextField "Campo de texto_10" at 199,33 size 215x43; Text 'Control Nivel'
   Button "Botón_7" at 617,698 size 130x48; TextOff 'Control Caudal'
      on Click: ActivateScreen("2_Control_Caudal", 0)

screen "6_Control_General" 1024x768
   GraphicView "Visor de gráficos_2" at 1,0 size 1023x766; Picture "Gráfico_22"
   GraphicView "Visor de gráficos_1" at 0,0 size 574x768; Picture "steven_tanque_png"
   Bar "Barra_1" at 261,226 size 72x397; MinimumValue 0; MaximumValue 300
      ProcessValue <- "LEVEL_METER_PANTALLA"
   Button "Botón_1" at 603,50 size 125x31; TextOff 'Start_Sistema'
      on Release: ResetBit("START_SISTEMA_HMI")
      on Press: SetBit("START_SISTEMA_HMI")
   Button "Botón_2" at 811,49 size 123x32; TextOff 'Stop_Sistema'
      on Release: ResetBit("STOP_SISTEMA_HMI")
      on Press: SetBit("STOP_SISTEMA_HMI")
   IOField "Campo ES_2" at 846,184 size 59x39; FormatPattern 999
      ProcessValue <- "DATA_INPUT_DISCHARGE_VALVE"
   TextField "Campo de texto_2" at 781,149 size 175x25; Text '% Válvula de Salida'
   Circle "Círculo_1" at 651,87 size 46x46
      Appearance <- "START_LIGHT"
   Circle "Círculo_2" at 846,88 size 45x45
      Appearance <- "STOP_LIGTH"
   TextField "Campo de texto_10" at 104,34 size 375x43; Text 'Control Caudal General'
   IOField "Campo ES_5" at 602,370 size 60x40; FormatPattern 999
      ProcessValue <- "PORCENT_CONEXION"
   IOField "Campo ES_6" at 601,425 size 61x40; FormatPattern 999
      ProcessValue <- "PORCENT_NIVEL"
   IOField "Campo ES_7" at 859,404 size 113x40
      ProcessValue <- "OUT_PID_FILL_VALVE_PID"
   GraphicView "Visor de gráficos_3" at 721,379 size 95x90; Picture "Gráfico_23"
   TextField "Campo de texto_5" at 582,464 size 53x25; Text 'Input'
   TextField "Campo de texto_6" at 898,373 size 65x25; Text 'Output'
   TextField "Campo de texto_7" at 596,345 size 78x25; Text 'Setpoint'
   IOField "Campo ES_3" at 651,184 size 60x40; FormatPattern 999
      ProcessValue <- "INPUT_SP_CAUDAL"
   TextField "Campo de texto_3" at 618,154 size 127x25; Text 'Valor SetPoint'
   IOField "Campo ES_1" at 605,551 size 60x40; FormatPattern 999
      ProcessValue <- "INPUT_SP_PID_CAUDAL"
   IOField "Campo ES_4" at 606,606 size 59x40; FormatPattern 999
      ProcessValue <- "CAUDAL_METER_PANTALLA"
   IOField "Campo ES_8" at 862,585 size 117x40
      ProcessValue <- "PORCENT_CONEXION"
   GraphicView "Visor de gráficos_4" at 721,560 size 98x90; Picture "Gráfico_23"
   TextField "Campo de texto_1" at 609,645 size 53x25; Text 'Input'
   TextField "Campo de texto_4" at 901,554 size 65x25; Text 'Output'
   TextField "Campo de texto_8" at 599,526 size 78x25; Text 'Setpoint'
   TextField "Campo de texto_9" at 674,301 size 217x43; Text 'Valores Nivel'
   TextField "Campo de texto_11" at 674,489 size 243x43; Text 'Valores Caudal'
   Switch "Interruptor_1" at 711,226 size 133x56; TextOn 'ON'; CaptionText 'Control PID'; TextOff 'OFF'
      ProcessValue <- "CONTROL_MANUAL"
   Button "Botón_5" at 762,697 size 116x50; TextOff 'Ir a Curvas'
      on Click: ActivateScreen("4_Curvas_Nivel", 0)
   Button "Botón_6" at 891,695 size 116x50; TextOff 'Ir a Inicio'
      on Click: ActivateScreen("1_Carátula", 0)
*)